# B&R Automation Studio project RobotNewEra (part 15)

### gmcipiec.cnc
```
Root (LangModule=ailgcode, Version=1.0)
  AxesSpec
  PrimTypes (PatternSuffix=:[^\d\w$#])
    BOOL (BRType=BOOL)
    STRING (BRType=STRING)
    WSTRING (BRType=WSTRING)
    TIME (BRType=TIME)
    SINT (BRType=SINT)
    INT (BRType=INT)
    DINT (BRType=DINT)
    USINT (BRType=USINT)
    UINT (BRType=UINT)
    UDINT (BRType=UDINT)
    REAL (BRType=REAL)
    LREAL (BRType=LREAL)
    DATE (BRType=DATE)
    DATE_AND_TIME (BRType=DATE_AND_TIME)
    DT (BRType=DT)
    TIME_OF_DAY (BRType=TIME_OF_DAY)
    TOD (BRType=TIME_OF_DAY)
    BYTE (BRType=BYTE)
    WORD (BRType=WORD)
    DWORD (BRType=DWORD)
  BuiltInProcs:
    SetCyclicId = #job->group_id = $[1]; (MinArgs=1, MaxArgs=1, Eval=Early)
    WaitForCyclic = if ( Defined(:$[1]:) ) 
        WaitForCyclicGroups(:${*}:);  
      else
        WaitForCyclicJob(:#last_job_id:);
      endif (MinArgs=0, MaxArgs=*)
    REPORT (MinArgs=2, MaxArgs=2)
      Arg (ref=id, DataType=INT)
      Arg (ref=msg, DataType=STRING)
    WARN (MinArgs=2, MaxArgs=2)
      Arg (ref=id, DataType=INT)
      Arg (ref=msg, DataType=STRING)
    HALT (MinArgs=2, MaxArgs=2)
      Arg (ref=id, DataType=INT)
      Arg (ref=msg, DataType=STRING)
    ERROR (MinArgs=2, MaxArgs=2)
      Arg (ref=id, DataType=INT)
      Arg (ref=msg, DataType=STRING)
    LOADBG (MinArgs=1, MaxArgs=1)
      Arg (ref=filename, DataType=STRING)
    LOAD (MinArgs=1, MaxArgs=1)
      Arg (ref=filename, DataType=STRING)
    UNLOAD (MinArgs=1, MaxArgs=1)
      Arg (ref=filename, DataType=STRING)
    EXEC (MinArgs=1, MaxArgs=3)
      Arg (ref=filename, DataType=STRING)
      Arg (ref=arguments, DataType=ANY_DATA)
      Arg (ref=langId, DataType=INT)
    EVAL = local $file_id;
      $file_id = LoadProgString(:$[1], $[2]:);
      WaitForLoadProg(:$file_id:);
      ExecProg(:$file_id:);
      UnloadProg(:$file_id:); (MinArgs=1, MaxArgs=2)
    PUSH_PACKET = PushPacket(::);
    PUSH_PACKET_CMD (MinArgs=1, MaxArgs=2)
      Arg (ref=cmd, DataType=INT)
      Arg (ref=data, DataType=ANY_DATA)
    DISPATCH_AND_WAIT (MinArgs=1, MaxArgs=1)
      Arg (ref=cmd, DataType=INT)
    START_PACKET_LIST = #inhibit_mp_list_dispatch = 1;
    END_PACKET_LIST = #inhibit_mp_list_dispatch = 0;
    LOG_INFO (MinArgs=1, MaxArgs=1)
      Arg (ref=msg, DataType=STRING)
    SET_BLOCK_NUMBER = SetCurBlockNr(:$[1]:); (MinArgs=1, MaxArgs=1)
    SBLOF_PATH = #next_motion.Command = MPCMD_SBL_PATH_INHIBIT;
      PushPacket(::);
    SBLON_PATH = #next_motion.Command = MPCMD_SBL_PATH_RELEASE;
      PushPacket(::);
  BuiltInFns:
    ABS = Abs(:$[1]:) (ReturnType=ANY_NUM, ArgType1=ANY_NUM, Inline=Yes)
    SIN = RSin(:$[1]:) (ReturnType=ANY_REAL, ArgType1=ANY_REAL, Inline=Yes)
    COS = RCos(:$[1]:) (ReturnType=ANY_REAL, ArgType1=ANY_REAL, Inline=Yes)
    TAN = RTan(:$[1]:) (ReturnType=ANY_REAL, ArgType1=ANY_REAL, Inline=Yes)
    ASIN = RASin(:$[1]:) (ReturnType=ANY_REAL, ArgType1=ANY_REAL, Inline=Yes)
    ACOS = RACos(:$[1]:) (ReturnType=ANY_REAL, ArgType1=ANY_REAL, Inline=Yes)
    ATAN = RATan(:$[1]:) (ReturnType=ANY_REAL, ArgType1=ANY_REAL, Inline=Yes)
    SQRT = Sqrt(:$[1]:) (ReturnType=ANY_REAL, ArgType1=ANY_REAL, Inline=Yes)
    LN = Ln(:$[1]:) (ReturnType=ANY_REAL, ArgType1=ANY_REAL, Inline=Yes)
    EXP = Exp(:$[1]:) (ReturnType=ANY_REAL, ArgType1=ANY_REAL, Inline=Yes)
    LOG = Log(:$[1]:) (ReturnType=ANY_REAL, ArgType1=ANY_REAL, Inline=Yes)
    EXPT = Pow(:$[1],$[2]:) (ReturnType=ANY_REAL, ArgType1=ANY_REAL, ArgType2=ANY_NUM, Inline=Yes)
    TRUNC = ToInt(:Fix(:$[1]:):) (ReturnType=IEC_INT, ArgType1=FLOAT, Inline=Yes)
    ADR = Adr(:\$[1]:) (ReturnType=IEC_UDINT, ArgType1=ANY_DATA, Inline=Yes)
    REF = \$[1] (ReturnType=ANY_DATA, ArgType1=ANY_DATA, Inline=Yes)
    SIZEOF = Sizeof(:\$[1]:) (ReturnType=IEC_UINT, NumArgs=1, Inline=Yes)
    LIMIT (ReturnType=ANY_NUM, Inline=No)
      Arg (ref=MIN, DataType=ANY_NUM)
      Arg (ref=IN, DataType=ANY_NUM)
      Arg (ref=MAX, DataType=ANY_NUM)
    MIN (ReturnType=ANY_NUM, Inline=No)
      Arg (ref=IN1, DataType=ANY_NUM)
      Arg (ref=IN2, DataType=ANY_NUM)
    MAX (ReturnType=ANY_NUM, Inline=No)
      Arg (ref=IN1, DataType=ANY_NUM)
      Arg (ref=IN2, DataType=ANY_NUM)
    ROL = BitRotL(:$[1],$[2]:) (ReturnType=ANY_NUM, ArgType1=ANY_NUM, ArgType2=IEC_SINT)
    ROR = BitRotR(:$[1],$[2]:) (ReturnType=ANY_NUM, ArgType1=ANY_NUM, ArgType2=IEC_SINT)
    SHR = BitShR(:$[1],$[2]:) (ReturnType=ANY_NUM, ArgType1=ANY_NUM, ArgType2=IEC_SINT)
    SHL = BitShL(:$[1],$[2]:) (ReturnType=ANY_NUM, ArgType1=ANY_NUM, ArgType2=IEC_SINT)
    BIT_TST = AsBitTst(:$[1],$[2]:) (ReturnType=ANY_NUM, ArgType1=ANY_NUM, ArgType2=IEC_SINT)
    BIT_SET = AsBitSet(:$[1],$[2]:) (ReturnType=ANY_NUM, ArgType1=ANY_NUM, ArgType2=IEC_SINT)
    BIT_CLR = AsBitClr(:$[1],$[2]:) (ReturnType=ANY_NUM, ArgType1=ANY_NUM, ArgType2=IEC_SINT)
    TO_BOOL = ToBool(:$[1]:) (ReturnType=IEC_BOOL, ArgType1=ANY_DATA, Inline=Yes)
    TO_USINT = ToUInt(:$[1],1:) (ReturnType=IEC_USINT, ArgType1=ANY_DATA, Inline=Yes)
    TO_BYTE = ToUInt(:$[1],1:) (ReturnType=IEC_BYTE, ArgType1=ANY_DATA, Inline=Yes)
    TO_SINT = ToInt(:$[1],1:) (ReturnType=IEC_SINT, ArgType1=ANY_DATA, Inline=Yes)
    TO_UINT = ToUInt(:$[1],2:) (ReturnType=IEC_UINT, ArgType1=ANY_DATA, Inline=Yes)
    TO_WORD = ToUInt(:$[1],2:) (ReturnType=IEC_WORD, ArgType1=ANY_DATA, Inline=Yes)
    TO_INT = ToInt(:$[1],2:) (ReturnType=IEC_INT, ArgType1=ANY_DATA, Inline=Yes)
    TO_UDINT = ToUInt(:$[1]:) (ReturnType=IEC_UDINT, ArgType1=ANY_DATA, Inline=Yes)
    TO_DWORD = ToUInt(:$[1]:) (ReturnType=IEC_DWORD, ArgType1=ANY_DATA, Inline=Yes)
    TO_DINT = ToInt(:$[1]:) (ReturnType=IEC_DINT, ArgType1=ANY_DATA, Inline=Yes)
    TO_TIME = ToTime(:$[1]:) (ReturnType=IEC_TIME, ArgType1=ANY_DATA, Inline=Yes)
    TO_DT = ToDT(:$[1]:) (ReturnType=IEC_DT, ArgType1=ANY_DATA, Inline=Yes)
    TO_DATE_AND_TIME = ToDT(:$[1]:) (ReturnType=IEC_DT, ArgType1=ANY_DATA, Inline=Yes)
    TO_TOD = ToTOD(:$[1]:) (ReturnType=IEC_TOD, ArgType1=ANY_DATA, Inline=Yes)
    TO_TIME_OF_DAY = ToTOD(:$[1]:) (ReturnType=IEC_TOD, ArgType1=ANY_DATA, Inline=Yes)
    TO_DATE = ToDate(:$[1]:) (ReturnType=IEC_DATE, ArgType1=ANY_DATA, Inline=Yes)
    TO_REAL = ToFloat(:$[1]:) (ReturnType=IEC_REAL, ArgType1=ANY_DATA, Inline=Yes)
    TO_LREAL = ToLReal(:$[1]:) (ReturnType=IEC_LREAL, ArgType1=ANY_DATA, Inline=Yes)
    TO_STRING = ToString(:$[1]:) (ReturnType=IEC_STRING, ArgType1=ANY_DATA, Inline=Yes)
    TO_WSTRING = ToWString(:$[1]:) (ReturnType=IEC_WSTRING, ArgType1=ANY_DATA, Inline=Yes)
    USINT_TO_BOOL = ToBool(:$[1]:) (ReturnType=IEC_BOOL, ArgType1=IEC_USINT, Inline=Yes)
    SINT_TO_BOOL = ToBool(:$[1]:) (ReturnType=IEC_BOOL, ArgType1=IEC_SINT, Inline=Yes)
    UINT_TO_BOOL = ToBool(:$[1]:) (ReturnType=IEC_BOOL, ArgType1=IEC_UINT, Inline=Yes)
    INT_TO_BOOL = ToBool(:$[1]:) (ReturnType=IEC_BOOL, ArgType1=IEC_INT, Inline=Yes)
    UDINT_TO_BOOL = ToBool(:$[1]:) (ReturnType=IEC_BOOL, ArgType1=IEC_UDINT, Inline=Yes)
    DINT_TO_BOOL = ToBool(:$[1]:) (ReturnType=IEC_BOOL, ArgType1=IEC_DINT, Inline=Yes)
    REAL_TO_BOOL = ToBool(:$[1]:) (ReturnType=IEC_BOOL, ArgType1=IEC_REAL, Inline=Yes)
    LREAL_TO_BOOL = ToBool(:$[1]:) (ReturnType=IEC_BOOL, ArgType1=IEC_LREAL, Inline=Yes)
    TIME_TO_BOOL = ToBool(:$[1]:) (ReturnType=IEC_BOOL, ArgType1=IEC_TIME, Inline=Yes)
    DT_TO_BOOL = ToBool(:$[1]:) (ReturnType=IEC_BOOL, ArgType1=IEC_DT, Inline=Yes)
    TOD_TO_BOOL = ToBool(:$[1]:) (ReturnType=IEC_BOOL, ArgType1=IEC_TOD, Inline=Yes)
    BYTE_TO_BOOL = ToBool(:$[1]:) (ReturnType=IEC_BOOL, ArgType1=IEC_BYTE, Inline=Yes)
    WORD_TO_BOOL = ToBool(:$[1]:) (ReturnType=IEC_BOOL, ArgType1=IEC_WORD, Inline=Yes)
    DWORD_TO_BOOL = ToBool(:$[1]:) (ReturnType=IEC_BOOL, ArgType1=IEC_DWORD, Inline=Yes)
    BOOL_TO_USINT = ToUInt(:$[1],1:) (ReturnType=IEC_USINT, ArgType1=IEC_BOOL, Inline=Yes)
    SINT_TO_USINT = ToUInt(:$[1],1:) (ReturnType=IEC_USINT, ArgType1=IEC_SINT, Inline=Yes)
    UINT_TO_USINT = ToUInt(:$[1],1:) (ReturnType=IEC_USINT, ArgType1=IEC_UINT, Inline=Yes)
    INT_TO_USINT = ToUInt(:$[1],1:) (ReturnType=IEC_USINT, ArgType1=IEC_INT, Inline=Yes)
    UDINT_TO_USINT = ToUInt(:$[1],1:) (ReturnType=IEC_USINT, ArgType1=IEC_UDINT, Inline=Yes)
    DINT_TO_USINT = ToUInt(:$[1],1:) (ReturnType=IEC_USINT, ArgType1=IEC_DINT, Inline=Yes)
    REAL_TO_USINT = ToUInt(:$[1],1:) (ReturnType=IEC_USINT, ArgType1=IEC_REAL, Inline=Yes)
    LREAL_TO_USINT = ToUInt(:$[1],1:) (ReturnType=IEC_USINT, ArgType1=IEC_LREAL, Inline=Yes)
    BOOL_TO_SINT = ToInt(:$[1],1:) (ReturnType=IEC_SINT, ArgType1=IEC_BOOL, Inline=Yes)
    USINT_TO_SINT = ToInt(:$[1],1:) (ReturnType=IEC_SINT, ArgType1=IEC_USINT, Inline=Yes)
    UINT_TO_SINT = ToInt(:$[1],1:) (ReturnType=IEC_SINT, ArgType1=IEC_UINT, Inline=Yes)
    INT_TO_SINT = ToInt(:$[1],1:) (ReturnType=IEC_SINT, ArgType1=IEC_INT, Inline=Yes)
    UDINT_TO_SINT = ToInt(:$[1],1:) (ReturnType=IEC_SINT, ArgType1=IEC_UDINT, Inline=Yes)
    DINT_TO_SINT = ToInt(:$[1],1:) (ReturnType=IEC_SINT, ArgType1=IEC_DINT, Inline=Yes)
    REAL_TO_SINT = ToInt(:$[1],1:) (ReturnType=IEC_SINT, ArgType1=IEC_REAL, Inline=Yes)
    LREAL_TO_SINT = ToInt(:$[1],1:) (ReturnType=IEC_SINT, ArgType1=IEC_LREAL, Inline=Yes)
    BOOL_TO_UINT = ToUInt(:$[1],2:) (ReturnType=IEC_UINT, ArgType1=IEC_BOOL, Inline=Yes)
    SINT_TO_UINT = ToUInt(:$[1],2:) (ReturnType=IEC_UINT, ArgType1=IEC_SINT, Inline=Yes)
    USINT_TO_UINT = ToUInt(:$[1],2:) (ReturnType=IEC_UINT, ArgType1=IEC_USINT, Inline=Yes)
    INT_TO_UINT = ToUInt(:$[1],2:) (ReturnType=IEC_UINT, ArgType1=IEC_INT, Inline=Yes)
    UDINT_TO_UINT = ToUInt(:$[1],2:) (ReturnType=IEC_UINT, ArgType1=IEC_UDINT, Inline=Yes)
    DINT_TO_UINT = ToUInt(:$[1],2:) (ReturnType=IEC_UINT, ArgType1=IEC_DINT, Inline=Yes)
    REAL_TO_UINT = ToUInt(:$[1],2:) (ReturnType=IEC_UINT, ArgType1=IEC_REAL, Inline=Yes)
    LREAL_TO_UINT = ToUInt(:$[1],2:) (ReturnType=IEC_UINT, ArgType1=IEC_LREAL, Inline=Yes)
    BOOL_TO_INT = ToInt(:$[1],2:) (ReturnType=IEC_INT, ArgType1=IEC_BOOL, Inline=Yes)
    SINT_TO_INT = ToInt(:$[1],2:) (ReturnType=IEC_INT, ArgType1=IEC_SINT, Inline=Yes)
    USINT_TO_INT = ToInt(:$[1],2:) (ReturnType=IEC_INT, ArgType1=IEC_USINT, Inline=Yes)
    UINT_TO_INT = ToInt(:$[1],2:) (ReturnType=IEC_INT, ArgType1=IEC_UINT, Inline=Yes)
    UDINT_TO_INT = ToInt(:$[1],2:) (ReturnType=IEC_INT, ArgType1=IEC_UDINT, Inline=Yes)
    DINT_TO_INT = ToInt(:$[1],2:) (ReturnType=IEC_INT, ArgType1=IEC_DINT, Inline=Yes)
    REAL_TO_INT = ToInt(:$[1],2:) (ReturnType=IEC_INT, ArgType1=IEC_REAL, Inline=Yes)
    LREAL_TO_INT = ToInt(:$[1],2:) (ReturnType=IEC_INT, ArgType1=IEC_LREAL, Inline=Yes)
    BOOL_TO_UDINT = ToUInt(:$[1]:) (ReturnType=IEC_UDINT, ArgType1=IEC_BOOL, Inline=Yes)
    USINT_TO_UDINT = ToUInt(:$[1]:) (ReturnType=IEC_UDINT, ArgType1=IEC_USINT, Inline=Yes)
    SINT_TO_UDINT = ToUInt(:$[1]:) (ReturnType=IEC_UDINT, ArgType1=IEC_SINT, Inline=Yes)
    UINT_TO_UDINT = ToUInt(:$[1]:) (ReturnType=IEC_UDINT, ArgType1=IEC_UINT, Inline=Yes)
    INT_TO_UDINT = ToUInt(:$[1]:) (ReturnType=IEC_UDINT, ArgType1=IEC_INT, Inline=Yes)
    DINT_TO_UDINT = ToUInt(:$[1]:) (ReturnType=IEC_UDINT, ArgType1=IEC_DINT, Inline=Yes)
    REAL_TO_UDINT = ToUInt(:$[1]:) (ReturnType=IEC_UDINT, ArgType1=IEC_REAL, Inline=Yes)
    LREAL_TO_UDINT = ToUInt(:$[1]:) (ReturnType=IEC_UDINT, ArgType1=IEC_LREAL, Inline=Yes)
    TIME_TO_UDINT = ToUInt(:$[1]:) (ReturnType=IEC_UDINT, ArgType1=IEC_TIME, Inline=Yes)
    DT_TO_UDINT = ToUInt(:$[1]:) (ReturnType=IEC_UDINT, ArgType1=IEC_DT, Inline=Yes)
    BOOL_TO_DINT = ToInt(:$[1]:) (ReturnType=IEC_DINT, ArgType1=IEC_BOOL, Inline=Yes)
    USINT_TO_DINT = ToInt(:$[1]:) (ReturnType=IEC_DINT, ArgType1=IEC_USINT, Inline=Yes)
    SINT_TO_DINT = ToInt(:$[1]:) (ReturnType=IEC_DINT, ArgType1=IEC_SINT, Inline=Yes)
    UINT_TO_DINT = ToInt(:$[1]:) (ReturnType=IEC_DINT, ArgType1=IEC_UINT, Inline=Yes)
    INT_TO_DINT = ToInt(:$[1]:) (ReturnType=IEC_DINT, ArgType1=IEC_INT, Inline=Yes)
    UDINT_TO_DINT = ToInt(:$[1]:) (ReturnType=IEC_DINT, ArgType1=IEC_UDINT, Inline=Yes)
    REAL_TO_DINT = ToInt(:$[1]:) (ReturnType=IEC_DINT, ArgType1=IEC_REAL, Inline=Yes)
    LREAL_TO_DINT = ToInt(:$[1]:) (ReturnType=IEC_DINT, ArgType1=IEC_LREAL, Inline=Yes)
    TIME_TO_DINT = ToInt(:$[1]:) (ReturnType=IEC_DINT, ArgType1=IEC_TIME, Inline=Yes)
    DT_TO_DINT = ToInt(:$[1]:) (ReturnType=IEC_DINT, ArgType1=IEC_DT, Inline=Yes)
    BOOL_TO_TIME = ToTime(:$[1]:) (ReturnType=IEC_TIME, ArgType1=IEC_BOOL, Inline=Yes)
    DINT_TO_TIME = ToTime(:$[1]:) (ReturnType=IEC_TIME, ArgType1=IEC_DINT, Inline=Yes)
    UDINT_TO_TIME = ToTime(:$[1]:) (ReturnType=IEC_TIME, ArgType1=IEC_UDINT, Inline=Yes)
    BOOL_TO_DT = ToDT(:$[1]:) (ReturnType=IEC_DT, ArgType1=IEC_BOOL, Inline=Yes)
    DINT_TO_DT = ToDT(:$[1]:) (ReturnType=IEC_DT, ArgType1=IEC_DINT, Inline=Yes)
    UDINT_TO_DT = ToDT(:$[1]:) (ReturnType=IEC_DT, ArgType1=IEC_UDINT, Inline=Yes)
    BOOL_TO_REAL = ToFloat(:$[1]:) (ReturnType=IEC_REAL, ArgType1=IEC_BOOL, Inline=Yes)
    USINT_TO_REAL = ToFloat(:$[1]:) (ReturnType=IEC_REAL, ArgType1=IEC_USINT, Inline=Yes)
    SINT_TO_REAL = ToFloat(:$[1]:) (ReturnType=IEC_REAL, ArgType1=IEC_SINT, Inline=Yes)
    UINT_TO_REAL = ToFloat(:$[1]:) (ReturnType=IEC_REAL, ArgType1=IEC_UINT, Inline=Yes)
    INT_TO_REAL = ToFloat(:$[1]:) (ReturnType=IEC_REAL, ArgType1=IEC_INT, Inline=Yes)
    UDINT_TO_REAL = ToFloat(:$[1]:) (ReturnType=IEC_REAL, ArgType1=IEC_UDINT, Inline=Yes)
    DINT_TO_REAL = ToFloat(:$[1]:) (ReturnType=IEC_REAL, ArgType1=IEC_DINT, Inline=Yes)
    LREAL_TO_REAL = ToFloat(:$[1]:) (ReturnType=IEC_REAL, ArgType1=IEC_LREAL, Inline=Yes)
    TIME_TO_REAL = ToFloat(:$[1]:) (ReturnType=IEC_REAL, ArgType1=IEC_TIME, Inline=Yes)
    BOOL_TO_LREAL = ToLReal(:$[1]:) (ReturnType=IEC_LREAL, ArgType1=IEC_BOOL, Inline=Yes)
    USINT_TO_LREAL = ToLReal(:$[1]:) (ReturnType=IEC_LREAL, ArgType1=IEC_USINT, Inline=Yes)
    SINT_TO_LREAL = ToLReal(:$[1]:) (ReturnType=IEC_LREAL, ArgType1=IEC_SINT, Inline=Yes)
    UINT_TO_LREAL = ToLReal(:$[1]:) (ReturnType=IEC_LREAL, ArgType1=IEC_UINT, Inline=Yes)
    INT_TO_LREAL = ToLReal(:$[1]:) (ReturnType=IEC_LREAL, ArgType1=IEC_INT, Inline=Yes)
    UDINT_TO_LREAL = ToLReal(:$[1]:) (ReturnType=IEC_LREAL, ArgType1=IEC_UDINT, Inline=Yes)
    DINT_TO_LREAL = ToLReal(:$[1]:) (ReturnType=IEC_LREAL, ArgType1=IEC_DINT, Inline=Yes)
    REAL_TO_LREAL = ToLReal(:$[1]:) (ReturnType=IEC_LREAL, ArgType1=IEC_REAL, Inline=Yes)
    TIME_TO_LREAL = ToLReal(:$[1]:) (ReturnType=IEC_LREAL, ArgType1=IEC_TIME, Inline=Yes)
    BOOL_TO_STRING = ToString(:ToBool(:$[1]:):) (ReturnType=IEC_STRING, ArgType1=IEC_BOOL, Inline=Yes)
    USINT_TO_STRING = ToString(:ToUInt(:$[1],1:):) (ReturnType=IEC_STRING, ArgType1=IEC_USINT, Inline=Yes)
    SINT_TO_STRING = ToString(:ToInt(:$[1],1:):) (ReturnType=IEC_STRING, ArgType1=IEC_SINT, Inline=Yes)
    UINT_TO_STRING = ToString(:ToUInt(:$[1],2:):) (ReturnType=IEC_STRING, ArgType1=IEC_UINT, Inline=Yes)
    INT_TO_STRING = ToString(:ToInt(:$[1],2:):) (ReturnType=IEC_STRING, ArgType1=IEC_INT, Inline=Yes)
    UDINT_TO_STRING = ToString(:ToUInt(:$[1]:):) (ReturnType=IEC_STRING, ArgType1=IEC_UDINT, Inline=Yes)
    DINT_TO_STRING = ToString(:ToInt(:$[1]:):) (ReturnType=IEC_STRING, ArgType1=IEC_DINT, Inline=Yes)
    REAL_TO_STRING = ToString(:ToFloat(:$[1]:):) (ReturnType=IEC_STRING, ArgType1=IEC_REAL, Inline=Yes)
    LREAL_TO_STRING = ToString(:ToLReal(:$[1]:):) (ReturnType=IEC_STRING, ArgType1=IEC_LREAL, Inline=Yes)
    STRING_TO_BOOL = ToBool(:StrToInt(:$[1]:):) (ReturnType=IEC_BOOL, ArgType1=IEC_STRING, Inline=Yes)
    STRING_TO_USINT = ToUInt(:StrToInt(:$[1]:),1:) (ReturnType=IEC_USINT, ArgType1=IEC_STRING, Inline=Yes)
    STRING_TO_SINT = ToInt(:StrToInt(:$[1]:),1:) (ReturnType=IEC_SINT, ArgType1=IEC_STRING, Inline=Yes)
    STRING_TO_UINT = ToUInt(:StrToInt(:$[1]:),2:) (ReturnType=IEC_UINT, ArgType1=IEC_STRING, Inline=Yes)
    STRING_TO_INT = ToInt(:StrToInt(:$[1]:),2:) (ReturnType=IEC_INT, ArgType1=IEC_STRING, Inline=Yes)
    STRING_TO_UDINT = ToUInt(:StrToInt(:$[1]:):) (ReturnType=IEC_UDINT, ArgType1=IEC_STRING, Inline=Yes)
    STRING_TO_DINT = ToInt(:StrToInt(:$[1]:):) (ReturnType=IEC_DINT, ArgType1=IEC_STRING, Inline=Yes)
    STRING_TO_REAL = ToFloat(:ToLReal(:$[1]:):) (ReturnType=IEC_REAL, ArgType1=IEC_STRING, Inline=Yes)
    STRING_TO_LREAL = ToLReal(:$[1]:) (ReturnType=IEC_LREAL, ArgType1=IEC_STRING, Inline=Yes)
    LEN = __LEN(:$[1]:) (ReturnType=IEC_INT, ArgType1=IEC_STRING, Inline=Yes)
    LEFT = __LEFT(:$[1], $[2]:) (ReturnType=IEC_STRING, ArgType1=IEC_STRING, ArgType2=IEC_INT, Inline=Yes)
    RIGHT = __RIGHT(:$[1], $[2]:) (ReturnType=IEC_STRING, ArgType1=IEC_STRING, ArgType2=IEC_INT, Inline=Yes)
    MID = __MID(:$[1], $[2], $[3]:) (ReturnType=IEC_STRING, ArgType1=IEC_STRING, ArgType2=IEC_INT, ArgType3=IEC_INT, Inline=Yes)
    CONCAT = __CONCAT(:$[1], $[2]:) (ReturnType=IEC_STRING, ArgType1=IEC_STRING, ArgType2=IEC_STRING, Inline=Yes)
    INSERT = __INSERT(:$[1], $[2], $[3]:) (ReturnType=IEC_STRING, ArgType1=IEC_STRING, ArgType2=IEC_STRING, ArgType3=IEC_INT, Inline=Yes)
    DELETE = __DELETE(:$[1], $[2], $[3]:) (ReturnType=IEC_STRING, ArgType1=IEC_STRING, ArgType2=IEC_INT, ArgType3=IEC_INT, Inline=Yes)
    REPLACE = __REPLACE(:$[1], $[2], $[3], $[4]:) (ReturnType=IEC_STRING, ArgType1=IEC_STRING, ArgType2=IEC_STRING, ArgType3=IEC_INT, ArgType4=IEC_INT, Inline=Yes)
    FIND = __FIND(:$[1], $[2]:) (ReturnType=IEC_INT, ArgType1=IEC_STRING, ArgType2=IEC_STRING, Inline=Yes)
    IP_INST_NUM = IpInstNum(::) (ReturnType=IEC_INT, NumArgs=0)
    IP_OWNER_ID = IpOwnerId(::) (ReturnType=IEC_INT, NumArgs=0)
    PACKET_DATA_ADR = GetIpInt(:6:) (ReturnType=IEC_UDINT, NumArgs=0, Inline=Yes)
    PACKET_COMMAND_ADR = GetIpInt(:7:) (ReturnType=IEC_UDINT, NumArgs=0, Inline=Yes)
  Parameters:
    QUOTED (QuotedName=$R, ValueType=FLOAT, ReturnType=IEC_LREAL)
      ARG (ref=EXPR, DataType=INT, MinValue=0, MaxValue=999)
    QUOTED (QuotedName=$P, ValueType=FLOAT, ReturnType=IEC_LREAL)
      ARG (ref=EXPR, DataType=INT, MinValue=0, MaxValue=999)
    QUOTED (QuotedName=$EXB, ValueType=INT, ReturnType=IEC_SINT)
      ARG (ref=EXPR, DataType=INT, MinValue=0, MaxValue=99)
    QUOTED (QuotedName=$EXW, ValueType=INT, ReturnType=IEC_INT)
      ARG (ref=EXPR, DataType=INT, MinValue=0, MaxValue=99)
    QUOTED (QuotedName=$EXL, ValueType=INT, ReturnType=IEC_DINT)
      ARG (ref=EXPR, DataType=INT, MinValue=0, MaxValue=99)
    QUOTED (QuotedName=$EXF, ValueType=FLOAT, ReturnType=IEC_REAL)
      ARG (ref=EXPR, DataType=INT, MinValue=0, MaxValue=3999)
    QUOTED (QuotedName=$MW, Synchronous=Yes, ValueType=INT, ReturnType=IEC_INT)
      ARG (ref=EXPR, DataType=INT, MinValue=0, MaxValue=99)
    QUOTED (QuotedName=$ML, Synchronous=Yes, ValueType=INT, ReturnType=IEC_DINT)
      ARG (ref=EXPR, DataType=INT, MinValue=0, MaxValue=99)
    QUOTED (QuotedName=$MF, Synchronous=Yes, ValueType=FLOAT, ReturnType=IEC_REAL)
      ARG (ref=EXPR, DataType=INT, MinValue=0, MaxValue=99)
  ParserData (NestedComments=No, DefaultCaseSensitive=Yes, CommentsSpanLines=Yes, ReadWholeFileBeforeParsing=Yes, ExpectMainProgStmts=No, UseFubTemplates=No, LexerType=IEC, RuntimePreventOverflow=No, RoundRealToInt=No, AllowArrayRefWithoutIndex=Yes, DeclareEnumLiteralsAsConstants=No, AllowVariableAutoDereference=Yes, AllowStructMemberAutoDereference=No, AllowPassByRefFnArgAutoReference=No, AllowNamedFnArgs=Yes, AllowUnnamedFnArgs=Yes, AllowFnArgMixedNaming=Yes, AllowFnArgsOutOfSequence=No, AllowBuiltinFnArgsOutOfSequence=Yes, AllowFnArgsOmmitted=Yes, AllowIgnoredFnReturn=Yes, AllowIgnoredExtraSubArgs=No, AllowFnStringInputArgsShort=No, RefuseBuiltinFnUnknownArgName=Yes, AllowBuiltinFnArgCaseSensitive=Yes)
    TKG_OPEN_COMMENT = (*
    TKG_CLOSE_COMMENT = *)
    TKG_IEC_LINE_COMMENT = //
    TKG_TRUE = TRUE:[^\w\d] (IsPattern=Yes)
    TKG_FALSE = FALSE:[^\w\d] (IsPattern=Yes)
    TKG_PRIM_TYPE (IsPattern=Yes)
    TKG_OPEN_BRACKET = (
    TKG_CLOSE_BRACKET = )
    TKG_OPEN_INDEXBRACKET = [
    TKG_CLOSE_INDEXBRACKET = ]
    TKG_COMMA = ,
    TKG_SUBRANGE = ..
    TKG_IEC_BINARY_INTEGER = 2#_[01][01_]+|2#[01][01_]+|2#_[01]|2#[01] (IsPattern=Yes)
    TKG_IEC_OCTAL_INTEGER = 8#_[0-7][0-7_]+|8#[0-7][0-7_]+|8#_[0-7]|8#[0-7] (IsPattern=Yes)
    TKG_IEC_HEX_INTEGER = 16#_[\da-fA-F][\da-fA-F]+|16#[\da-fA-F][\da-fA-F_]+|16#_[\da-fA-F]|16#[\da-fA-F] (IsPattern=Yes)
    TKG_REAL = \d[\d_]*\.[\d_]+[Ee][\+\-]\d[\d_]*|\d[\d_]*\.[\d_]+[Ee]\d[\d_]*|\d[\d_]*\.[\d_]+ (IsPattern=Yes)
    TKG_REAL_EXP = \d[\d_]*[Ee]\d[\d_]*|\d[\d_]*[Ee][\+\-]\d[\d_]* (IsPattern=Yes)
    TKG_INTEGER = \d|\d[\d_]+ (IsPattern=Yes)
    TKG_DOT = .
    TKG_PATHSYNCH_REC_IEC = DO_PATH_SYNCH:[^\w\d] (IsPattern=Yes, EndRuleToken=Yes)
    TKG_PATHSYNCH_END = END_PATH_SYNCH:[^\w\d] (IsPattern=Yes, EndRuleToken=Yes)
    TKG_PATHSYNCH_IPEVAL = IP_EVAL:[^\w\d] (IsPattern=Yes)
    TKG_CYCLIC_PATHSYNCH_BLOCKING_IEC = CYCLIC_PS_BL:[^\w\d] (IsPattern=Yes, EndRuleToken=Yes)
    TKG_CYCLIC_PATHSYNCH_IEC = CYCLIC_PS:[^\w\d] (IsPattern=Yes, EndRuleToken=Yes)
    TKG_CYCLIC_BLOCKING_IEC = CYCLIC_BL:[^\w\d] (IsPattern=Yes, EndRuleToken=Yes)
    TKG_CYCLIC_IEC = CYCLIC:[^\w\d] (IsPattern=Yes, EndRuleToken=Yes)
    TKG_CYCLIC_END_IEC = END_CYCLIC:[^\w\d] (IsPattern=Yes, EndRuleToken=Yes)
    TKG_REFERENCE = REFERENCE:[^\w\d] (FollowedBy=TKG_IEC_TO, IsPattern=Yes)
    TKG_IEC_TO = TO:[^\w\d] (IsPattern=Yes)
    TKG_IEC_DO = DO:[^\w\d] (IsPattern=Yes, EndRuleToken=Yes)
    TKG_FOR_NOFINALDEC = FOR:[^\w\d] (FileXLInvalid=Yes, IsPattern=Yes)
    TKG_FORSTEP = BY:[^\w\d] (FileXLInvalid=Yes, IsPattern=Yes)
    TKG_ENDFOR = END_FOR:[^\w\d] (FileXLInvalid=Yes, IsPattern=Yes, EndRuleToken=Yes)
    TKG_IF = IF:[^\w\d] (IsPattern=Yes)
    TKG_THEN = THEN:[^\w\d] (IsPattern=Yes, EndRuleToken=Yes)
    TKG_BLOCK_ELSEIF = ELSIF:[^\w\d] (IsPattern=Yes)
    TKG_ELSE_AND_DEFAULT = ELSE:[^\w\d] (IsPattern=Yes, EndRuleToken=Yes)
    TKG_BLOCK_ENDIF = END_IF:[^\w\d] (IsPattern=Yes, EndRuleToken=Yes)
    TKG_SWITCH = CASE:[^\w\d] (IsPattern=Yes, FileXLInvalid=Yes)
    TKG_ENDSWITCH_NOBREAK = END_CASE:[^\w\d] (FileXLInvalid=Yes, IsPattern=Yes, EndRuleToken=Yes)
    TKG_WHILE = WHILE:[^\w\d] (FileXLInvalid=Yes, IsPattern=Yes)
    TKG_ENDWHILE = END_WHILE:[^\w\d] (FileXLInvalid=Yes, IsPattern=Yes, EndRuleToken=Yes)
    TKG_DO = REPEAT:[^\w\d] (FileXLInvalid=Yes, IsPattern=Yes, EndRuleToken=Yes)
    TKG_ENDDO_UNTIL = UNTIL:[^\w\d] (FileXLInvalid=Yes, IsPattern=Yes)
    TKG_ENDDO_POSTCOND = END_REPEAT:[^\w\d] (FileXLInvalid=Yes, IsPattern=Yes, EndRuleToken=Yes)
    TKG_BREAK = EXIT:[^\w\d] (FileXLInvalid=Yes, IsPattern=Yes)
    TKG_RETURN = RETURN:[^\w\d] (FileXLInvalid=Yes, IsPattern=Yes)
    TKG_IEC_SEL_FN = SEL:[^\w\d] (FileXLInvalid=Yes, IsPattern=Yes)
    TKG_IEC_MUX_FN = MUX:[^\w\d] (FileXLInvalid=Yes, IsPattern=Yes)
    TKG_TIME_LITERAL = time#\-[dDhHmMsS_\.\d]+|time#[dDhHmMsS_\.\d]+|t#\-[dDhHmMsS_\.\d]+|t#[dDhHmMsS_\.\d]+ (CaseSensitive=no, IsPattern=yes)
    TKG_DATE_AND_TIME_LITERAL = DT#[12]\d\d\d\-[\d\:\-]*|DATE_AND_TIME#[12]\d\d\d\-[\d\:\-]* (CaseSensitive=no, IsPattern=yes)
    TKG_DATE_LITERAL = D#[12]\d\d\d\-[\d\-]*|DATE#[12]\d\d\d\-[\d\-]* (CaseSensitive=no, IsPattern=yes)
    TKG_TIME_OF_DAY_LITERAL = TOD#\d[\d\:\.]*|TIME_OF_DAY#\d[\d\:\.]* (CaseSensitive=no, IsPattern=yes)
    TKG_ASSIGN_EQ = :=
    TKG_OPEN_IP_EXTENSION = {
    TKG_CLOSE_IP_EXTENSION = }
    TKG_IEC_OPEN_TYPE = TYPE:[^\w\d] (IsPattern=Yes)
    TKG_IEC_CLOSE_TYPE = END_TYPE:[^\w\d] (IsPattern=Yes, EndRuleToken=Yes)
    TKG_VAR = VAR:[^\w\d] (IsPattern=Yes)
    TKG_VAR_GLOBAL = VAR_GLOBAL:[^\w\d] (IsPattern=Yes)
    TKG_VAR_INPUT = VAR_INPUT:[^\w\d] (IsPattern=Yes)
    TKG_VAR_OUTPUT = VAR_OUTPUT:[^\w\d] (IsPattern=Yes)
    TKG_VAR_IN_OUT = VAR_IN_OUT:[^\w\d] (IsPattern=Yes)
    TKG_VAR_END = END_VAR:[^\w\d] (IsPattern=Yes, EndRuleToken=Yes)
    TKG_VAR_RETAIN = RETAIN:[^\d\w] (IsPattern=Yes)
    TKG_IP_RETAIN = IP_RETAIN:[^\d\w] (IsPattern=Yes)
    TKG_AT = AT:[^\d\w] (IsPattern=Yes)
    TKG_PLC = PLC:[^\d\w] (IsPattern=Yes)
    TKG_PV_UNDECL = UNRETAIN_VAR:[^\d\w] (IsPattern=Yes)
    TKG_VARSYNCH_IP = IP_SYNCH:[^\d\w] (IsPattern=Yes)
    TKG_VARSYNCH_PATH = PATH_SYNCH:[^\d\w] (IsPattern=Yes)
    TKG_CONSTANT = CONSTANT:[^\d\w] (IsPattern=Yes)
    TKG_VARSCOPE_IP_GLOBAL = IP_GLOBAL:[^\w\d] (IsPattern=Yes)
    TKG_VARSCOPE_SHARED_IP_GLOBAL = SHARED_IP_GLOBAL:[^\w\d] (IsPattern=Yes)
    TKG_VARSCOPE_NC_GLOBAL = NC_GLOBAL:[^\w\d] (IsPattern=Yes)
    TKG_VARSCOPE_PLC_GLOBAL = PLC_GLOBAL:[^\w\d] (IsPattern=Yes)
    TKG_VARSCOPE_IP_LOCAL = LOCAL:[^\w\d] (IsPattern=Yes)
    TKG_IEC_DATATYPE_SPEC = : (IsPattern=No)
    TKG_IEC_ARRAY = ARRAY:[^\w\d] (IsPattern=Yes)
    TKG_IEC_OF = OF:[^\w\d] (IsPattern=Yes)
    TKG_IEC_DELIM = ; (EndRuleToken=Yes)
    TKG_IEC_OPEN_STRUCT = STRUCT:[^\w\d] (IsPattern=Yes)
    TKG_IEC_CLOSE_STRUCT = END_STRUCT:[^\w\d] (IsPattern=Yes)
    TKG_BITWISE_LP_BINARY_AND = AND:[^\w\d] (IsPattern=Yes)
    TKG_BITWISE_LP_BINARY_OR = OR:[^\w\d] (IsPattern=Yes)
    TKG_BITWISE_LP_BINARY_XOR = XOR:[^\w\d] (IsPattern=Yes)
    TKG_BITWISE_UNARY_COMPLEMENT = NOT:[^\w\d] (IsPattern=Yes)
    TKG_COMP_EXACT_BINARY_GREATER_THAN_OR_EQ = >=
    TKG_COMP_EXACT_BINARY_LESS_THAN_OR_EQ = <=
    TKG_COMP_EXACT_BINARY_EQUAL_TO = =
    TKG_COMP_EXACT_BINARY_NOT_EQUAL_TO = <>
    TKG_COMP_EXACT_BINARY_GREATER_THAN = >
    TKG_COMP_EXACT_BINARY_LESS_THAN = <
    TKG_ARITH_BINARY_PLUS = +
    TKG_ARITH_BINARY_MINUS = -
    TKG_ARITH_BINARY_POWER = **
    TKG_ARITH_BINARY_MULTIPLY = *
    TKG_ARITH_BINARY_DIVIDE = /
    TKG_ARITH_BINARY_MODULO = MOD:[^\w\d] (IsPattern=Yes)
    TKG_PRAGMA = #pragma:[^\w\d] (IsPattern=Yes, FollowedBy=TKG_IDENTIFIER)
    TKG_INCLUDE = #include:[^\w\d] (IsPattern=Yes)
    TKG_PROG_START = PROGRAM:[^\w\d] (IsPattern=Yes, FollowedBy=TKG_PROG_NAME)
    TKG_PROG_NAME = _INIT:[^\w\d]|_CYCLIC:[^\w\d]|_EXIT:[^\w\d]|_MAIN:[^\w\d] (IsPattern=Yes, EndRuleToken=Yes)
    TKG_PROG_END = END_PROGRAM:[^\w\d] (IsPattern=Yes, EndRuleToken=Yes)
    TKG_SUBPROG_START = FUNCTION:[^\w\d] (IsPattern=Yes)
    TKG_SUBPROG_END = END_FUNCTION:[^\w\d] (IsPattern=Yes, EndRuleToken=Yes)
    TKG_FUB_DECL = FUNCTION_BLOCK:[^\w\d] (IsPattern=Yes)
    TKG_FUB_END = END_FUNCTION_BLOCK:[^\w\d] (IsPattern=Yes, EndRuleToken=Yes)
    TKG_RETURN = RETURN:[^\w\d] (IsPattern=Yes)
    TKG_ACCESS = ACCESS:[^\w\d] (IsPattern=Yes)
    TKG_DEREF_OP = ^
    TKG_ACTION = ACTION:[^\w\d] (IsPattern=Yes)
    TKG_ACTION_END = END_ACTION:[^\w\d] (IsPattern=Yes, EndRuleToken=Yes)
    TKG_IEC_TYPED_VALUE = \w#:[\w\d\+\-]|\w[\w\d]+#:[\w\d\+\-] (IsPattern=Yes)
    TKG_PARAM_PREFIX = $R:[^\w\d]|$P:[^\w\d]|$MW:[^\w\d]|$ML:[^\w\d]|$MF:[^\w\d]|$EXW:[^\w\d]|$EXL:[^\w\d]|$EXF:[^\w\d]|$EXB:[^\w\d] (IsPattern=Yes)
    TKG_IDENTIFIER = \w|\w[\w\d$]+|$[\w\d$]+ (IsPattern=Yes)
    TKG_INIT_IDENTIFIER = \w|\w[\w\d$]+|$[\w\d$]+ (IsPattern=Yes, Disabled=Yes)
  StringChars (AsciiStringStart=', AsciiStringEnd=', UTF16StringStart=", UTF16StringEnd=")
    EscapeSeq (Search=$N, CaseSensitive=Yes, ReplaceValue=10)
    EscapeSeq (Search=$n, CaseSensitive=Yes, ReplaceValue=10)
    EscapeSeq (Search=$L, CaseSensitive=Yes, ReplaceValue=10)
    EscapeSeq (Search=$l, CaseSensitive=Yes, ReplaceValue=10)
    EscapeSeq (Search=$P, CaseSensitive=Yes, ReplaceValue=12)
    EscapeSeq (Search=$p, CaseSensitive=Yes, ReplaceValue=12)
    EscapeSeq (Search=$R, CaseSensitive=Yes, ReplaceValue=13)
    EscapeSeq (Search=$r, CaseSensitive=Yes, ReplaceValue=13)
    EscapeSeq (Search=$T, CaseSensitive=Yes, ReplaceValue=9)
    EscapeSeq (Search=$t, CaseSensitive=Yes, ReplaceValue=9)
    EscapeSeq (Search=$', CaseSensitive=Yes, ReplaceStr=')
    EscapeSeq (Search=$", CaseSensitive=Yes, ReplaceStr=")
    EscapeSeq (Search=$[\dA-Fa-f]+, IsPattern=Yes, CaseSensitive=Yes, ReplaceEncodingBase=16)
    EscapeSeq (Search=$$, ReplaceStr=$)
    EscapeSeq (Search=$, ReplaceStr=)
```

- Data object Logical/GmcIpConfig/gmciplbr (Cnc, version 2.48.1) (no source held here)

- Data object Logical/GmcIpConfig/gmciplsm (Cnc, version 2.48.1) (no source held here)

- Data object Logical/GmcIpConfig/gmcipmx (Cnc, version 2.48.1) (no source held here)

- Data object Logical/GmcIpConfig/gmcipmxd (Cnc, version 2.48.1) (no source held here)

### gmcipfub.cnc
```
CONFIG:
  FUBOutputs
  FUBS
```

- Data object Logical/GmcIpUserConfig/gmcipfun (Cnc, version 2.48.1) (no source held here)

- Data object Logical/GmcIpUserConfig/gmcipubr (Cnc, version 2.48.1) (no source held here)

- Data object Logical/GmcIpUserConfig/gmcipuc (Cnc, version 2.48.1) (no source held here)

- Data object Logical/GmcIpUserConfig/gmcipus (Cnc, version 2.48.1) (no source held here)

- Data object Logical/GmcIpUserConfig/gmcipvar (Cnc, version 2.48.1) (no source held here)

### Program Logical/test (ANSIC)

#### Main.cpp - Init, cyclic, exit code
```cpp
#include <bur/plctypes.h>

#ifdef _DEFAULT_INCLUDES
	#include <AsDefault.h>
#endif

// amount of memory to be allocated for heap storage must be specified for every ANSI C++ program with the bur_heap_size variable
unsigned long bur_heap_size = 0xFFFF;

void _INIT ProgramInit(void)
{
	// Insert code here
	int i=0;

}

void _CYCLIC ProgramCyclic(void)
{
	// Insert code here
	i++;
}

void _EXIT ProgramExit(void)
{
	// Insert code here

}
```

Listed in the project but not available here: Logical/MotionHandling/FeedForward/OptMotConfig.typ, Logical/HmiHandling/HmiMain/HmiFile/HmiFileLocal.var, Logical/HmiHandling/HmiEditor/HmiFileVar/HmiFileVarLocal.typ, Logical/test/Types.typ, Logical/test/Variables.var
